Staubli VAL3: onF6Event.pgx

program onF6Event()
  local string l_sPaste
  local bool l_bUndo
  local num l_nResult
begin
  // look if the bButton is enable
  if bButton[5]
    //
    //  Duplicate
    //
    l_sPaste=sEvent
    call alreadyExist(l_sPaste,l_bUndo)
    if !l_bUndo
      call trajType:duplicate(sEvent,l_sPaste,l_nResult)
      if l_nResult==0
        logMsg("[KERNEL] INTERFACE:Duplicate the trajectory: "+sEvent+" to: "+l_sPaste)
        sEvent=l_sPaste
        // update the memory stack
        call buildList()
      else
        popUpMsg("error code duplicate: "+toString("",l_nResult))
        logMsg("[KERNEL] INTERFACE:Duplicate the trajectory: "+sEvent+" to: "+l_sPaste+"errorCode"+toString("",l_nResult))
      endIf
    endIf
  endIf
end
